FUNCTION_BLOCK DateTime_TEST EXTENDS TcUnit.FB_TestSuite

CheckStringFormat();

METHOD CheckStringFormat
VAR_INST
  sut : DateTime;
  expected : STRING;
  result : STRING;
END_VAR
VAR
  localSystemTime : Tc2_Utilities.TIMESTRUCT;
END_VAR
sut();

TEST('CheckStringFormat');

localSystemTime := sut.AsLocalSystemTime;

expected := Tc2_Standard.CONCAT('-', TO_STRING(localSystemTime.wYear));
IF localSystemTime.wMonth < 10 THEN expected := Tc2_Standard.CONCAT(expected, '0'); END_IF
expected := Tc2_Standard.CONCAT(expected, TO_STRING(localSystemTime.wMonth));
IF localSystemTime.wDay < 10 THEN expected := Tc2_Standard.CONCAT(expected, '0'); END_IF
expected := Tc2_Standard.CONCAT(expected, TO_STRING(localSystemTime.wDay));
expected := Tc2_Standard.CONCAT(expected, '-');
IF localSystemTime.wHour < 10 THEN expected := Tc2_Standard.CONCAT(expected, '0'); END_IF
expected := Tc2_Standard.CONCAT(expected, TO_STRING(localSystemTime.wHour));
expected := Tc2_Standard.CONCAT(expected, ':');
IF localSystemTime.wMinute < 10 THEN expected := Tc2_Standard.CONCAT(expected, '0'); END_IF
expected := Tc2_Standard.CONCAT(expected, TO_STRING(localSystemTime.wMinute));
expected := Tc2_Standard.CONCAT(expected, ':');
IF localSystemTime.wSecond < 10 THEN expected := Tc2_Standard.CONCAT(expected, '0'); END_IF
expected := Tc2_Standard.CONCAT(expected, TO_STRING(localSystemTime.wSecond));
expected := Tc2_Standard.CONCAT(expected, '-');

result := sut.ToFormatString('-YYYYMMDD-hh:mm:ss-');
  
IF sut.Done THEN
  AssertEquals(
    Expected  :=  expected,
    Actual    :=  result,
    Message   :=  'Time formatting failed.'
  );

  TEST_FINISHED();
END_IF
END_METHOD

END_FUNCTION_BLOCK

(* stored: Version 1.1.0.1
   POU DateTime_TEST: Id {5cec2056-1949-4f6f-b2b8-e6d4752d21ea}, SpecialFunc None
   Method CheckStringFormat: Id {eeedfcd3-9548-4730-bde7-8f00a6d4c7e6} *)
